(* IEC 61131-3 sources: CodesysTest/export/Pro24.dev/Plc Logic/Application, 5 files *)

(* ---- Globals.gvl.st ---- *)
(*#-#-#-#-#-#-#-#-#-#---Declaration---#-#-#-#-#-#-#-#-#-#-#-#-#*)

{attribute 'qualified_only'}
VAR_GLOBAL
    firstScan : BOOL; //First Scan Bit
    STEPS_PER_INCH : INT;  //Steps Per Inch for Pressure Bar Servos
    enableDryCycle : BOOL;          // Enable dry cycle
	SystemLog : FB_InternalLogger;
	jawMovingIn : BOOL;
	passthroughChangedFromJog : BOOL;
	machinePowerOK : BOOL;
END_VAR

VAR_GLOBAL CONSTANT
    STEPS_PER_INCH_SEAL_FLATTENER_HORIZONTAL_AXIS_MOTOR  : INT := 2500;
    STEPS_PER_INCH_SEAL_FLATTENER_VERTICAL_AXIS_MOTOR : INT := 2890;        //Steps per inch for NEMA 17 seal flattener finger motor
    STEPS_PER_INCH_BIG_MOTOR : INT := 21872;        //Steps per inch for NEMA 17 motor
    STEPS_PER_INCH_SMALL_MOTOR : INT := 19600;        //Steps per inch for NEMA 11 motor
    STEPS_PER_INCH_SHOW_MOTOR : INT := 18900;        //Steps per inch for NEMA 11 motor
    STEPS_PER_INCH_PRINTER : INT := 4498;            //Steps per inch for printer step servo
    STEPS_PER_INCH_20_DEGREE_BAG_DELIVERY : INT := 5093; // Steps per inch for 20 degree bag delivery motors
	STEPS_PER_INCH_ADJUSTABLE_PASSTHROUGH : INT := 19530;  // Steps per inch for the Adjustable Passthrough motor
	STEPS_PER_INCH_TFBelt : INT := 6833;  // Steps per inch for the Adjustable Passthrough motor
	STEPS_PER_INCH_TFLS : INT := 10000;  // Steps per inch for the Adjustable Passthrough motor
    VELOCITY_IPS_MULTIPLIER_20_DEGREE_BAG_DELIVERY: REAL := 61;
    PASSTHROUGH_ZERO_OFFSET : REAL := 2;            //Zero offset for passthough (minimum passthough)
    MAX_BAG_WIDTH : REAL := 18;                //Passthrough setting
	AMP_MOTOR_RPI : INT := 10;
	MAX_LOGGED_ITEMS : UINT := 500;	// Max items to be logged
	IO_MASTER_INPUT_BYTES : INT := 64;
	IO_MASTER_OUTPUT_BYTES : INT := 22;
	MAX_VALVE_MANIFOLD_STATIONS : UINT := 12;
END_VAR

VAR_GLOBAL
    headCycleCount : DINT;                 // Head Cycle Counts
	headCycleCount2 : DINT;                 // Head Cycle Counts
    bagGrabberCycleCount : DINT;         // Bag Grabber Cycle Counts
    solenoidCycleCount1 : DINT;         // Solenoid Cycle Cycle Counts (first solenoid)
    motorizedSealFlattenersCount : DINT;         // MSF Cycle Counts
    bagOpenFingersCount : DINT;        // Bag Open Finger Cycles
    sealFlattenerFingersCount : DINT;  // Seal Flattener Fingers Cycle Count
    electricPressureBarCount : DINT;    // Electric Pressure bar Cycle count
    sealBarCount : DINT;                 // Seal bar Cycle count
    bagDeliveryCycleCount : DINT;        // Bag Delivery Cycle Count
    printerCycleCounts : DINT;            // Printer Cycle Counts
    bagsMadeCount : DINT;                // Bags Made
    passthroughChangeCount : DINT;        // Passthrough Changes
	passthroughChangeDistance : UDINT;	// Passthrough Distance Changes in .1 Inches
	solenoidCycleCount2 : DINT;     	// Solenoid Cycle Cycle Counts (Strech SX)
	solenoidFailureCount2 : UDINT;		// Solenoid Failure Count (Strech SX)
	pickAndPlaceCycleCount : UDINT;		// Pick and place cycle count
	passthroughChangeCount2 : DINT;        // Passthrough Changes
	passthroughChangeDistance2 : UDINT;	// Passthrough Distance Changes in .1 Inches
	bagFailedToGrabBothFingersCount : UDINT; // Both Fingers failed to grab bag
	bagFailedToGrabRightFingerCount : UDINT; // Right Bag Open Finger Failed to Grab Bag
	bagFailedToGrabLeftFingerCount : UDINT; // Left Bag Open Finger Failed to Grab Bag
	successfulBagOpenCount : UDINT;			// Successful Bag Open Count
	rejectedBagCount : UDINT;				// Rejected bag count
    dryCycleCount  :UDINT;                   // Dry cycle count
	lastPrinterDelta : TIME := T#100MS;
	factoryTestComplete : BOOL;		// 1000 bags test done
END_VAR

(* ---- IO.gvl.st ---- *)
(*#-#-#-#-#-#-#-#-#-#---Declaration---#-#-#-#-#-#-#-#-#-#-#-#-#*)

{attribute 'qualified_only'}
{attribute 'FBVisuCreator'}
{attribute 'global_init_slot' := '50010'}
VAR_GLOBAL
	iPressureBarExtended : FB_PhysicalDigitalInput(name := 'Pressure Bar Open Prox') := (in := Devices.IOMaster.headIONode.iPort0Pin2);
	iPressureBarRetracted : FB_PhysicalDigitalInput(name := 'Pressure Bar Closed Prox') := (in := Devices.IOMaster.headIONode.iPort0Pin4);
	iPressureBarNotObstructed : FB_PhysicalDigitalInput(name := 'Pressure Bar Not Obstructed Input') := (in := Devices.IOMaster.headIONode.iPort1Pin2);
	iBagPhotoeyeClear : FB_PhysicalDigitalInput(name := 'Bag Edge Photoeye Clear') := (in := Devices.IOMaster.headIONode.iPort1Pin4);
	iBagOpenFingersRightBagPresent : FB_PhysicalDigitalInput(name := 'Right BOF Bag Present') := (in := Devices.IOMaster.headIONode.iPort2Pin2);
	iBagOpenFingersLeftBagPresent : FB_PhysicalDigitalInput(name := 'Left BOF Bag Present') := (in := Devices.IOMaster.headIONode.iPort2Pin4);
	iPowerOnButton : FB_PhysicalDigitalInput(name := 'Power On Button Input') := (in := Devices.IOMaster.headIONode.iPort3Pin2);
	oPowerOnIndication : FB_PhysicalDigitalOutput(name := 'Power On Indication Lamp') := (refOutput := Devices.IOMaster.headIONode.oPort3Pin4);
	//iUnwindBagLevel : FB_PhysicalAnalogInput(name := 'Unwind Bag Level') := (in := Devices.IOMaster.headIONode.iIOLinkPort4);
	iSealBarExtended : FB_PhysicalDigitalInput(name := 'Seal Bar Extended Prox') := (in := Devices.IOMaster.headIONode.iPort5Pin2);
	{warning 'TODO: Seal bar temp is actually iolinkport5 but is faked out for now because of Murr bug'}
	iSealBarTemperature : FB_PhysicalAnalogInput(name := 'Seal Bar Temperature') := (in := Devices.IOMaster.headIONode.iIOLinkPort4, enableLogging := TRUE, logDeadband := 20);
	iMachineInitiateCycle : FB_PhysicalDigitalInput(name := 'Machine Initiate Cycle Input') := (in := Devices.IOMaster.headIONode.iPort6Pin2);
	//iFunnelHighSpeedCounter : FB_PhysicalAnalogInput(name := 'Funnel Parts Count') := (in := Devices.IOMaster.headIONode.iIOLinkPort6);
	iMCROn : FB_PhysicalDigitalInput(name := 'MCR On Input') := (in := Devices.IOMaster.headIONode.iPort7Pin2);

	iPrinterDataReady : FB_PhysicalDigitalInput(name := 'Printer Data Ready Signal') := (in := Devices.IOMaster.printerIONode.iX000);
	iPrinterEndOfPrint : FB_PhysicalDigitalInput(name := 'Printer End Print Signal') := (in := Devices.IOMaster.printerIONode.iX001);
	iPrinterServiceRequired : FB_PhysicalDigitalInput(name := 'Printer Service Required Signal') := (in := Devices.IOMaster.printerIONode.iX002);
	iPrinterRibbonOut : FB_PhysicalDigitalInput(name := 'Printer Ribbon Out Signal') := (in := Devices.IOMaster.printerIONode.iX003);
	oPrinterStartPrint : FB_PhysicalDigitalOutput(name := 'Printer Start Print Signal') := (refOutput := Devices.IOMaster.printerIONode.oX100);
	oRunRibbonUnwindMotor : FB_PhysicalDigitalOutput(name := 'Run Ribbon Unwind') := (refOutput := Devices.IOMaster.printerIONode.oX101);;

	iFunnelOpened : FB_PhysicalDigitalInput(name := 'Funnel Opened Prox') := (in := Devices.IOMaster.frontGuardIONode.iPort0Pin2);
	iFunnelClosed : FB_PhysicalDigitalInput(name := 'Funnel Closed Prox') := (in := Devices.IOMaster.frontGuardIONode.iPort0Pin4);
	iLDunkLowered : FB_PhysicalDigitalInput(name := 'L-Dunk Lowered Prox') := (in := Devices.IOMaster.frontGuardIONode.iPort1Pin2);
	iLDunkRaised : FB_PhysicalDigitalInput(name := 'L-Dunk Raised Prox') := (in := Devices.IOMaster.frontGuardIONode.iPort1Pin4);
	iAccumFunnelOpened : FB_PhysicalDigitalInput(name := 'Accumulating Funnel Opened') := (in := Devices.IOMaster.frontGuardIONode.iPort2Pin2);
	iAccumFunnelClosed : FB_PhysicalDigitalInput(name := 'Accumulating Funnel Closed') := (in := Devices.IOMaster.frontGuardIONode.iPort2Pin4);
	iPalmButtonRightActive : FB_PhysicalDigitalInput(name := 'Right Palm Button Activated') := (in := Devices.IOMaster.frontGuardIONode.iPort3Pin2);
	iPalmButtonLeftActive : FB_PhysicalDigitalInput(name := 'Left Palm Button Activated') := (in := Devices.IOMaster.frontGuardIONode.iPort3Pin4);

	iLoadPlateInLoadingPosition :  FB_PhysicalDigitalInput(name := 'Load Plate in Loading Position Prox') := (in := Devices.IOMaster.dischargeIONode.iPort0Pin2);
	iLoadPlateInDischargePosition : FB_PhysicalDigitalInput(name := 'Load Plate in Discharge Position Prox') := (in := Devices.IOMaster.dischargeIONode.iPort0Pin4);
	iLoadShelfInLoadingPosition : FB_PhysicalDigitalInput(name := 'Load Shelf in Loading Position Prox') := (in := Devices.IOMaster.dischargeIONode.iPort1Pin2);
	iLoadShelfInDischargePosition : FB_PhysicalDigitalInput(name := 'Load Shelf in Loading Position Prox') := (in := Devices.IOMaster.dischargeIONode.iPort1Pin4);
	oExitConveyorRunCommand : FB_PhysicalDigitalOutput(name := 'Exit Conveyor Run Command') := (refOutput := Devices.IOMaster.dischargeIONode.oPort2Pin2);
	iExitConveyorRunningFeedback : FB_PhysicalDigitalInput(name := 'Exit Conveyor Running') := (in := Devices.IOMaster.dischargeIONode.iPort2Pin4);
	iDischargeProductClear : FB_PhysicalDigitalInput(name := 'Product Clear Sensor') := (in := Devices.IOMaster.dischargeIONode.iPort3Pin2);
	oSoftStartEnable : FB_PhysicalDigitalOutput(name := 'Soft Start Enable Solenoid') := (refOutput := Devices.IOMaster.dischargeIONode.oPort4Pin4);

	iFillerTrigger : BOOL;
	iFillerOK : BOOL;
	iBaggerInhibit : BOOL;
	oBaggerOK : BOOL;
	oReadyForFiller : BOOL;
	oWaitingForPrinter : BOOL;
	(*
	oExtendPressureBarCylinder : FB_PhysicalDigitalOutput(name := 'Extend Pressure Bar Solenoid') := (refOutput := Devices.valveManifold.oValve0Solenoid0);;
	oRetractPressureBarCylinder : FB_PhysicalDigitalOutput(name := 'Retract Pressure Bar Solenoid') := (refOutput := Devices.valveManifold.oValve0Solenoid1);;
	oRetractLoadPlateCylinder : BOOL;
	oOpenHPAValve : BOOL;
	oOpenLPAValve : BOOL;
	oExtendSealBarCylinder : BOOL;
	oExtendPrintHeadCylinder : BOOL;
	oRotateBOFUp : FB_PhysicalDigitalOutput(name := 'Rotate BOF Up Solenoid') := (refOutput := Devices.valveManifold.oValve3Solenoid0);
	oRotateBOFDown : FB_PhysicalDigitalOutput(name := 'Rotate BOF Down Solenoid') := (refOutput := Devices.valveManifold.oValve3Solenoid1);
	*)
END_VAR

(* ---- Devices.pou.st ---- *)
(*#-#-#-#-#-#-#-#-#-#---Declaration---#-#-#-#-#-#-#-#-#-#-#-#-#*)

PROGRAM Devices
VAR

END_VAR
VAR_IN_OUT

END_VAR

VAR_OUTPUT

	IOMaster : FB_MurrMaster(name := 'IO Master') := 	(ptrEIPInputs := ADR(IOEIPInputs),
														 ptrEIPOutputs := ADR(IOEIPOutputs));

	pressureBarSolenoidValve : FB_DoubleSolenoidOpenCenterActuator(name := 'Pressure Bar SV');
	sealBarSolenoidValve : FB_SingleSolenoidNormallyRetractedActuator(name := 'Seal Bar SV');
	HPA_LPA_SolenoidValve : FB_DoubleSolenoidClosedCenterActuator(name := 'HPA/LPA SV');
	loadPlateSolenoidValve : FB_DoubleSolenoidOpenCenterActuator(name := 'Load Plate SV');
	bagOpenFingersSolenoidValve : FB_DoubleSolenoidOpenCenterActuator(name := 'BOF SV');
	printHeadSolenoidValve : FB_SingleSolenoidNormallyRetractedActuator(name := 'Print Head SV');
	vacuumSolenoidValve : FB_VacuumGenerator(name := 'Vacuum SV');
	sealFlattenersVertAxisSolenoidValve : FB_DoubleSolenoidOpenCenterActuator(name := 'Seal Flattener Vert SV');
	loadShelfSolenoidValve : FB_DoubleSolenoidOpenCenterActuator(name := 'Load Shelf SV');
	blankSolenoidValve : FB_SolenoidValve(name := 'Blank SV');
	i : UINT;

	valveManifold : FB_SolenoidValveManifold(name := 'Valve Manifold') := (ptrEIPOutputs := ADR(Valve_Manifold_Outputs));

END_VAR
(*#-#-#-#-#-#-#-#-#-#---Implementation---#-#-#-#-#-#-#-#-#-#-#-#-#*)

// Valve manifold station selection
FOR i := 1 TO Globals.MAX_VALVE_MANIFOLD_STATIONS DO
	CASE HMIData.stationValveSelection[i] OF

		ValveSelection.PressureBar : 						valveManifold.station[i] := pressureBarSolenoidValve;

		ValveSelection.SealBar : 							valveManifold.station[i] := sealBarSolenoidValve;

		ValveSelection.HPA_LPA : 							valveManifold.station[i] := HPA_LPA_SolenoidValve;

		ValveSelection.LoadPlate : 							valveManifold.station[i] := loadPlateSolenoidValve;

		ValveSelection.BagOpenFingers : 					valveManifold.station[i] := bagOpenFingersSolenoidValve;

		ValveSelection.PrintHead : 							valveManifold.station[i] := printHeadSolenoidValve;

		ValveSelection.Vacuum : 							valveManifold.station[i] := vacuumSolenoidValve;

		ValveSelection.SealFlattenersVerticalAxis : 		valveManifold.station[i] := sealFlattenersVertAxisSolenoidValve;

		ValveSelection.LoadShelf : 							valveManifold.station[i] := loadShelfSolenoidValve;

		ValveSelection.Blank : 								valveManifold.station[i] := blankSolenoidValve;

	ELSE
		valveManifold.station[i] := blankSolenoidValve;
	END_CASE
END_FOR

// Run all configured valves and then the manifold
pressureBarSolenoidValve();
sealBarSolenoidValve();
HPA_LPA_SolenoidValve();
loadPlateSolenoidValve();
bagOpenFingersSolenoidValve();
printHeadSolenoidValve();
vacuumSolenoidValve();
sealFlattenersVertAxisSolenoidValve();
loadShelfSolenoidValve();
blankSolenoidValve();
valveManifold();

IOMaster();

(* ---- IOUpdatePOU.pou.st ---- *)
(*#-#-#-#-#-#-#-#-#-#---Declaration---#-#-#-#-#-#-#-#-#-#-#-#-#*)

PROGRAM IOUpdatePOU
VAR
END_VAR
(*#-#-#-#-#-#-#-#-#-#---Implementation---#-#-#-#-#-#-#-#-#-#-#-#-#*)

(* ---- PLC_PRG.pou.st ---- *)
(*#-#-#-#-#-#-#-#-#-#---Declaration---#-#-#-#-#-#-#-#-#-#-#-#-#*)

PROGRAM PLC_PRG
VAR_INPUT
END_VAR
VAR_OUTPUT
END_VAR
VAR
END_VAR
(*#-#-#-#-#-#-#-#-#-#---Implementation---#-#-#-#-#-#-#-#-#-#-#-#-#*)
